FUNCTION_BLOCK CmdSludgeDischargeSLBLogic (* CAT Function Block Type *)
  (* Standard: 61499-2 *)
  (* Version 4.1, 9/30/2026, Claude/Hidryco, Schneider Electric, Rev4.1 - Velocidade reenviada a cada mudanca de comando das bombas e a cada 1 s (SpeedGate aberto); Rev4 - PID pela logica; Rev3.1 - SpeedGate *)
  PACKAGE SE.Nereda;
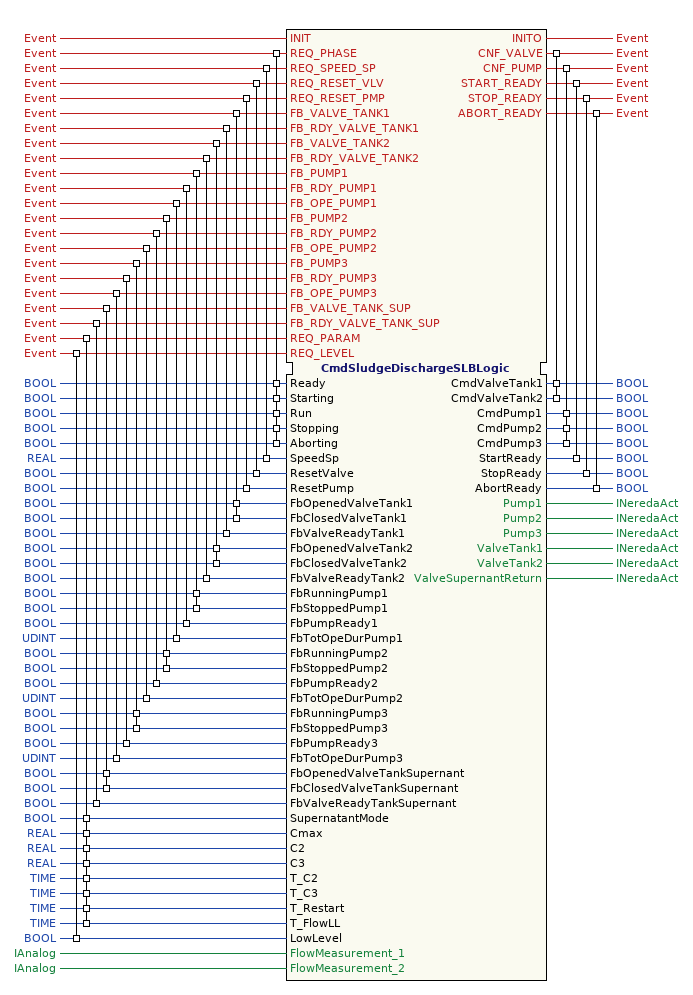
  EVENT_INPUT
    INIT;
    REQ_PHASE WITH Ready, Starting, Run, Stopping, Aborting;
    REQ_SPEED_SP WITH SpeedSp;
    REQ_RESET_VLV WITH ResetValve;
    REQ_RESET_PMP WITH ResetPump;
    FB_VALVE_TANK1 WITH FbOpenedValveTank1, FbClosedValveTank1;
    FB_RDY_VALVE_TANK1 WITH FbValveReadyTank1;
    FB_VALVE_TANK2 WITH FbOpenedValveTank2, FbClosedValveTank2;
    FB_RDY_VALVE_TANK2 WITH FbValveReadyTank2;
    FB_PUMP1 WITH FbRunningPump1, FbStoppedPump1;
    FB_RDY_PUMP1 WITH FbPumpReady1;
    FB_OPE_PUMP1 WITH FbTotOpeDurPump1;
    FB_PUMP2 WITH FbRunningPump2, FbStoppedPump2;
    FB_RDY_PUMP2 WITH FbPumpReady2;
    FB_OPE_PUMP2 WITH FbTotOpeDurPump2;
    FB_PUMP3 WITH FbRunningPump3, FbStoppedPump3;
    FB_RDY_PUMP3 WITH FbPumpReady3;
    FB_OPE_PUMP3 WITH FbTotOpeDurPump3;
    FB_VALVE_TANK_SUP WITH FbOpenedValveTankSupernant, FbClosedValveTankSupernant;
    FB_RDY_VALVE_TANK_SUP WITH FbValveReadyTankSupernant;
    REQ_PARAM WITH SupernatantMode, Cmax, C2, C3, T_C2, T_C3, T_Restart, T_FlowLL; (* Parametros da logica de bombas e da pausa *)
    REQ_LEVEL WITH LowLevel; (* Nivel L do 49LT0001 *)
  END_EVENT
  EVENT_OUTPUT
    INITO;
    CNF_VALVE WITH CmdValveTank1, CmdValveTank2;
    CNF_PUMP WITH CmdPump1, CmdPump2, CmdPump3;
    START_READY WITH StartReady;
    STOP_READY WITH StopReady;
    ABORT_READY WITH AbortReady;
  END_EVENT
  VAR_INPUT
    Ready : BOOL;
    Starting : BOOL;
    Run : BOOL;
    Stopping : BOOL;
    Aborting : BOOL;
    SpeedSp : REAL;
    ResetValve : BOOL;
    ResetPump : BOOL;
    FbOpenedValveTank1 : BOOL;
    FbClosedValveTank1 : BOOL;
    FbValveReadyTank1 : BOOL;
    FbOpenedValveTank2 : BOOL;
    FbClosedValveTank2 : BOOL;
    FbValveReadyTank2 : BOOL;
    FbRunningPump1 : BOOL;
    FbStoppedPump1 : BOOL;
    FbPumpReady1 : BOOL;
    FbTotOpeDurPump1 : UDINT;
    FbRunningPump2 : BOOL;
    FbStoppedPump2 : BOOL;
    FbPumpReady2 : BOOL;
    FbTotOpeDurPump2 : UDINT;
    FbRunningPump3 : BOOL;
    FbStoppedPump3 : BOOL;
    FbPumpReady3 : BOOL;
    FbTotOpeDurPump3 : UDINT;
    FbOpenedValveTankSupernant : BOOL;
    FbClosedValveTankSupernant : BOOL;
    FbValveReadyTankSupernant : BOOL;
    SupernatantMode : BOOL; (* TRUE = sobrenadante (2 servico + 1 reserva); FALSE/desligado = lodo (1 servico + 2 reserva) *)
    Cmax : REAL; (* Vazao maxima de 1 bomba [m3/h] *)
    C2 : REAL; (* Vazao por bomba na entrada da 2a bomba [m3/h] *)
    C3 : REAL; (* Vazao por bomba abaixo da qual sai 1 bomba [m3/h] *)
    T_C2 : TIME; (* Tempo em C2 *)
    T_C3 : TIME; (* Tempo abaixo de C3 *)
    T_Restart : TIME; (* Pausa: tempo para retomar *)
    T_FlowLL : TIME; (* Vazao LL por este tempo com bomba rodando = pausa (0 = desabilitado) *)
    LowLevel : BOOL; (* Nivel L do 49LT0001 (pausa a descarga) *)
  END_VAR
  VAR_OUTPUT
    CmdValveTank1 : BOOL;
    CmdValveTank2 : BOOL;
    CmdPump1 : BOOL;
    CmdPump2 : BOOL;
    CmdPump3 : BOOL;
    StartReady : BOOL;
    StopReady : BOOL;
    AbortReady : BOOL;
  END_VAR
  SOCKETS
    FlowMeasurement_1 : IAnalog;
  END_SOCKETS
  SOCKETS
    FlowMeasurement_2 : IAnalog;
  END_SOCKETS
  PLUGS
    Pump1 : INeredaAct;
    Pump2 : INeredaAct;
    Pump3 : INeredaAct;
    ValveTank1 : INeredaAct;
    ValveTank2 : INeredaAct;
    ValveSupernantReturn : INeredaAct;
  END_PLUGS
  (* 01 - FUNCTIONNAL INPUT INTERFACE *)
  (* 00 - INITIALIZATION *)
  (* 05 - LOGIC *)
  (* 06 - HMI INTERFACE *)
  (* 03 - FIELD INTERFACE *)
  (* 02 - FUNCTIONNAL OUTPUT INTERFACE *)
  (* Command Logic *)
  (* SIGNAL SELECTION *)
  FBS
    CmdLogic : CmdSludgeDischargeSLBLogicBasic;
    ValveCmdSmoothTank1 : boolValueChanged;
    PumpCmdSmooth1 : boolValueChanged;
    FbOpenValveTank1 : DS_SELECTX_2536758B411A6CE51; {SET_ATTRIBUTE(Configuration.GenericFBType.InterfaceParams, Runtime.Standard#CNTX:=2;CNTY:=1;DI${CNTX,_,CNTY$}:BOOL)}
    FbCloseValveTank1 : DS_SELECTX_2536758B411A6CE51; {SET_ATTRIBUTE(Configuration.GenericFBType.InterfaceParams, Runtime.Standard#CNTX:=2;CNTY:=1;DI${CNTX,_,CNTY$}:BOOL)}
    FbRunPump1 : DS_SELECTX_2536758B411A6CE51; {SET_ATTRIBUTE(Configuration.GenericFBType.InterfaceParams, Runtime.Standard#CNTX:=2;CNTY:=1;DI${CNTX,_,CNTY$}:BOOL)}
    FbStopPump1 : DS_SELECTX_2536758B411A6CE51; {SET_ATTRIBUTE(Configuration.GenericFBType.InterfaceParams, Runtime.Standard#CNTX:=2;CNTY:=1;DI${CNTX,_,CNTY$}:BOOL)}
    FbReadyPump1 : DS_SELECTX_2536758B411A6CE51; {SET_ATTRIBUTE(Configuration.GenericFBType.InterfaceParams, Runtime.Standard#CNTX:=2;CNTY:=1;DI${CNTX,_,CNTY$}:BOOL)}
    FbReadyValveTank1 : DS_SELECTX_2536758B411A6CE51; {SET_ATTRIBUTE(Configuration.GenericFBType.InterfaceParams, Runtime.Standard#CNTX:=2;CNTY:=1;DI${CNTX,_,CNTY$}:BOOL)}
    ValveCmdTank1 : BOOL2INT;
    PumpCmd1 : BOOL2INT;
    FbTotOpePump1 : DS_SELECTX_29841900CAFD143A; {SET_ATTRIBUTE(Configuration.GenericFBType.InterfaceParams, Runtime.Standard#CNTX:=2;CNTY:=1;DI${CNTX,_,CNTY$}:UDINT)}
    FbRunPump2 : DS_SELECTX_2536758B411A6CE51; {SET_ATTRIBUTE(Configuration.GenericFBType.InterfaceParams, Runtime.Standard#CNTX:=2;CNTY:=1;DI${CNTX,_,CNTY$}:BOOL)}
    FbStopPump2 : DS_SELECTX_2536758B411A6CE51; {SET_ATTRIBUTE(Configuration.GenericFBType.InterfaceParams, Runtime.Standard#CNTX:=2;CNTY:=1;DI${CNTX,_,CNTY$}:BOOL)}
    FbReadyPump2 : DS_SELECTX_2536758B411A6CE51; {SET_ATTRIBUTE(Configuration.GenericFBType.InterfaceParams, Runtime.Standard#CNTX:=2;CNTY:=1;DI${CNTX,_,CNTY$}:BOOL)}
    FbTotOpePump2 : DS_SELECTX_29841900CAFD143A; {SET_ATTRIBUTE(Configuration.GenericFBType.InterfaceParams, Runtime.Standard#CNTX:=2;CNTY:=1;DI${CNTX,_,CNTY$}:UDINT)}
    FbRunPump3 : DS_SELECTX_2536758B411A6CE51; {SET_ATTRIBUTE(Configuration.GenericFBType.InterfaceParams, Runtime.Standard#CNTX:=2;CNTY:=1;DI${CNTX,_,CNTY$}:BOOL)}
    FbStopPump3 : DS_SELECTX_2536758B411A6CE51; {SET_ATTRIBUTE(Configuration.GenericFBType.InterfaceParams, Runtime.Standard#CNTX:=2;CNTY:=1;DI${CNTX,_,CNTY$}:BOOL)}
    FbReadyPump3 : DS_SELECTX_2536758B411A6CE51; {SET_ATTRIBUTE(Configuration.GenericFBType.InterfaceParams, Runtime.Standard#CNTX:=2;CNTY:=1;DI${CNTX,_,CNTY$}:BOOL)}
    FbTotOpePump3 : DS_SELECTX_29841900CAFD143A; {SET_ATTRIBUTE(Configuration.GenericFBType.InterfaceParams, Runtime.Standard#CNTX:=2;CNTY:=1;DI${CNTX,_,CNTY$}:UDINT)}
    FbOpenValveTank2 : DS_SELECTX_2536758B411A6CE51; {SET_ATTRIBUTE(Configuration.GenericFBType.InterfaceParams, Runtime.Standard#CNTX:=2;CNTY:=1;DI${CNTX,_,CNTY$}:BOOL)}
    FbCloseValveTank2 : DS_SELECTX_2536758B411A6CE51; {SET_ATTRIBUTE(Configuration.GenericFBType.InterfaceParams, Runtime.Standard#CNTX:=2;CNTY:=1;DI${CNTX,_,CNTY$}:BOOL)}
    FbReadyValveTank2 : DS_SELECTX_2536758B411A6CE51; {SET_ATTRIBUTE(Configuration.GenericFBType.InterfaceParams, Runtime.Standard#CNTX:=2;CNTY:=1;DI${CNTX,_,CNTY$}:BOOL)}
    ValveCmdSmoothTank2 : boolValueChanged;
    ValveCmdTank2 : BOOL2INT;
    PumpCmdSmooth2 : boolValueChanged;
    PumpCmd2 : BOOL2INT;
    PumpCmdSmooth3 : boolValueChanged;
    PumpCmd3 : BOOL2INT;
    MergeValveCmd : E_MERGE;
    MergePumpCmd : E_MERGE;
    IThis : CmdSludgeDischargeSLBLogic_HMI(QI := TRUE);
    PID : PID; {SET_ATTRIBUTE(Configuration.Component.HideUnusedPorts, )}
    PIDISc : PID_Manager;
    SpeedSp1 : SpeedSpFlowSensorFail;
    Flow_Status : decodeStatus; {SET_ATTRIBUTE(Configuration.Component.HideUnusedPorts, )}
    OR1 : OR_550FE6D62F509EB3; {SET_ATTRIBUTE(Configuration.GenericFBType.InterfaceParams, Runtime.Standard#CNT:=3;OUT:BOOL)}
    PumpCmdSmooth4 : boolValueChanged;
    PumpCmd4 : BOOL2INT;
    FbOpenValveTankSupernant : DS_SELECTX_2536758B411A6CE51; {SET_ATTRIBUTE(Configuration.GenericFBType.InterfaceParams, Runtime.Standard#CNTX:=2;CNTY:=1;DI${CNTX,_,CNTY$}:BOOL)}
    FbCloseValveTankSupernant : DS_SELECTX_2536758B411A6CE51; {SET_ATTRIBUTE(Configuration.GenericFBType.InterfaceParams, Runtime.Standard#CNTX:=2;CNTY:=1;DI${CNTX,_,CNTY$}:BOOL)}
    FbReadyValveTankSupernant : DS_SELECTX_2536758B411A6CE51; {SET_ATTRIBUTE(Configuration.GenericFBType.InterfaceParams, Runtime.Standard#CNTX:=2;CNTY:=1;DI${CNTX,_,CNTY$}:BOOL)}
    TickCycle : E_CYCLE(DT := T#1s);
    SpeedGate : E_PERMIT;
  END_FBS
  EVENT_CONNECTIONS
    FbOpenValveTank1.CNF1 TO FbCloseValveTank1.REQ1;
    FbOpenValveTank1.CNF2 TO FbCloseValveTank1.REQ2;
    FbRunPump1.CNF1 TO FbStopPump1.REQ1;
    FbRunPump1.CNF2 TO FbStopPump1.REQ2;
    ValveCmdSmoothTank1.CHD TO ValveCmdTank1.DD5870AA881150BB;
    PumpCmdSmooth1.CHD TO PumpCmd1.DD5870AA881150BB;
    FB_VALVE_TANK1 TO FbOpenValveTank1.REQ2;
    FB_PUMP1 TO FbRunPump1.REQ2;
    FB_RDY_VALVE_TANK1 TO FbReadyValveTank1.REQ2;
    FB_RDY_PUMP1 TO FbReadyPump1.REQ2;
    REQ_PHASE TO CmdLogic.READY;
    REQ_PHASE TO CmdLogic.STARTING;
    REQ_PHASE TO CmdLogic.RUN;
    REQ_PHASE TO CmdLogic.STOPPING;
    REQ_PHASE TO CmdLogic.ABORTING;
    FbCloseValveTank1.IND TO CmdLogic.VALVE_FB_OPEN;
    FbStopPump1.IND TO CmdLogic.PUMP_FB_RUN;
    FbReadyValveTank1.IND TO CmdLogic.VALVE_AVAILABLE;
    FbReadyPump1.IND TO CmdLogic.PUMP_NO_AVAILABLE;
    CmdLogic.VALVE_CNF TO ValveCmdSmoothTank1.REQ;
    CmdLogic.PUMP_CNF TO PumpCmdSmooth1.REQ;
    CmdLogic.START_READY TO START_READY;
    CmdLogic.STOP_READY TO STOP_READY;
    CmdLogic.ABORTED_READY TO ABORT_READY;
    FbRunPump2.CNF1 TO FbStopPump2.REQ1;
    FbRunPump2.CNF2 TO FbStopPump2.REQ2;
    FbRunPump3.CNF1 TO FbStopPump3.REQ1;
    FbRunPump3.CNF2 TO FbStopPump3.REQ2;
    FbOpenValveTank2.CNF1 TO FbCloseValveTank2.REQ1;
    FbOpenValveTank2.CNF2 TO FbCloseValveTank2.REQ2;
    ValveCmdSmoothTank2.CHD TO ValveCmdTank2.DD5870AA881150BB;
    PumpCmdSmooth2.CHD TO PumpCmd2.DD5870AA881150BB;
    PumpCmdSmooth3.CHD TO PumpCmd3.DD5870AA881150BB;
    FbReadyValveTank2.IND TO CmdLogic.VALVE_AVAILABLE;
    FbCloseValveTank2.IND TO CmdLogic.VALVE_FB_OPEN;
    FbTotOpePump1.IND TO CmdLogic.51724FB542235B99;
    FbTotOpePump3.IND TO CmdLogic.51724FB542235B99;
    FbTotOpePump2.IND TO CmdLogic.51724FB542235B99;
    FbStopPump3.IND TO CmdLogic.PUMP_FB_RUN;
    FbStopPump2.IND TO CmdLogic.PUMP_FB_RUN;
    FbReadyPump2.IND TO CmdLogic.PUMP_NO_AVAILABLE;
    FbReadyPump3.IND TO CmdLogic.PUMP_NO_AVAILABLE;
    FB_RDY_VALVE_TANK2 TO FbReadyValveTank2.REQ2;
    FB_VALVE_TANK2 TO FbOpenValveTank2.REQ2;
    FB_RDY_PUMP3 TO FbReadyPump3.REQ2;
    FB_OPE_PUMP3 TO FbTotOpePump3.REQ2;
    FB_PUMP3 TO FbRunPump3.REQ2;
    FB_RDY_PUMP2 TO FbReadyPump2.REQ2;
    FB_OPE_PUMP2 TO FbTotOpePump2.REQ2;
    FB_PUMP2 TO FbRunPump2.REQ2;
    ValveTank1.CC753684FA882790 TO FbReadyValveTank1.REQ1;
    ValveTank1.9CD053F8408797ED TO FbOpenValveTank1.REQ1;
    ValveTank2.9CD053F8408797ED TO FbOpenValveTank2.REQ1;
    ValveTank2.CC753684FA882790 TO FbReadyValveTank2.REQ1;
    Pump1.2DA8AEC15204E92D TO FbTotOpePump1.REQ1;
    Pump1.CC753684FA882790 TO FbReadyPump1.REQ1;
    Pump1.9CD053F8408797ED TO FbRunPump1.REQ1;
    FB_OPE_PUMP1 TO FbTotOpePump1.REQ2;
    Pump2.9CD053F8408797ED TO FbRunPump2.REQ1;
    Pump2.CC753684FA882790 TO FbReadyPump2.REQ1;
    Pump2.2DA8AEC15204E92D TO FbTotOpePump2.REQ1;
    Pump3.9CD053F8408797ED TO FbRunPump3.REQ1;
    Pump3.CC753684FA882790 TO FbReadyPump3.REQ1;
    Pump3.2DA8AEC15204E92D TO FbTotOpePump3.REQ1;
    ValveCmdTank1.6FC99A5BD1C38561 TO ValveTank1.0F1CDF9A9B4A227A;
    ValveCmdTank2.6FC99A5BD1C38561 TO ValveTank2.0F1CDF9A9B4A227A;
    PumpCmd1.6FC99A5BD1C38561 TO Pump1.0F1CDF9A9B4A227A;
    PumpCmd2.6FC99A5BD1C38561 TO Pump2.0F1CDF9A9B4A227A;
    PumpCmd3.6FC99A5BD1C38561 TO Pump3.0F1CDF9A9B4A227A;
    CmdLogic.PUMP_CNF TO PumpCmdSmooth3.REQ;
    CmdLogic.PUMP_CNF TO PumpCmdSmooth2.REQ;
    CmdLogic.VALVE_CNF TO ValveCmdSmoothTank2.REQ;
    REQ_RESET_VLV TO Pump3.37BBC1F841739733;
    REQ_RESET_VLV TO Pump1.37BBC1F841739733;
    REQ_RESET_VLV TO Pump2.37BBC1F841739733;
    ValveCmdSmoothTank1.CHD TO MergeValveCmd.EI1;
    ValveCmdSmoothTank2.CHD TO MergeValveCmd.EI2;
    MergeValveCmd.EO TO CNF_VALVE;
    PumpCmdSmooth1.CHD TO MergePumpCmd.EI1;
    PumpCmdSmooth2.CHD TO MergePumpCmd.EI2;
    PumpCmdSmooth3.CHD TO MergePumpCmd.EI2;
    MergePumpCmd.EO TO CNF_PUMP;
    PIDISc.CE80458C9D5EF15A TO INITO;
    FlowMeasurement_1.REQ TO Flow_Status.REQ;
    PumpCmdSmooth3.CHD TO OR1.REQ;
    PumpCmdSmooth2.CHD TO OR1.REQ;
    PumpCmdSmooth1.CHD TO OR1.REQ;
    OR1.CNF TO PIDISc.REQ;
    FlowMeasurement_1.REQ TO SpeedSp1.B5D6B08FA2666F02;
    INIT TO IThis.2F65FBA3287455C1;
    CmdLogic.001688431DB935DE TO IThis.2568B13DF8BCDE7D;
    IThis.FFFD39D6E5C086B9 TO PIDISc.INIT;
    Flow_Status.CNF TO SpeedSp1.B5D6B08FA2666F02;
    PumpCmdSmooth4.CHD TO PumpCmd4.DD5870AA881150BB;
    PumpCmd4.6FC99A5BD1C38561 TO ValveSupernantReturn.0F1CDF9A9B4A227A;
    CmdLogic.VALVE_CNF TO PumpCmdSmooth4.REQ;
    FbOpenValveTankSupernant.CNF1 TO FbCloseValveTankSupernant.REQ1;
    FbOpenValveTankSupernant.CNF2 TO FbCloseValveTankSupernant.REQ2;
    ValveSupernantReturn.CC753684FA882790 TO FbReadyValveTankSupernant.REQ2;
    ValveSupernantReturn.9CD053F8408797ED TO FbOpenValveTankSupernant.REQ2;
    FB_VALVE_TANK_SUP TO FbOpenValveTankSupernant.REQ1;
    FB_RDY_VALVE_TANK_SUP TO FbReadyValveTankSupernant.REQ1;
    FbReadyValveTankSupernant.IND TO CmdLogic.VALVE_AVAILABLE;
    FbCloseValveTankSupernant.IND TO CmdLogic.VALVE_FB_OPEN;
    REQ_RESET_PMP TO ValveSupernantReturn.37BBC1F841739733;
    IThis.FFFD39D6E5C086B9 TO TickCycle.START;
    TickCycle.EO TO CmdLogic.2AFCCC4D006C5A58;
    REQ_SPEED_SP TO CmdLogic.888C7FFA93152C07;
    REQ_PARAM TO CmdLogic.888C7FFA93152C07;
    CmdLogic.948C0A3C8D4A59E4 TO PIDISc.REQ;
    CmdLogic.948C0A3C8D4A59E4 TO SpeedSp1.B5D6B08FA2666F02;
    REQ_LEVEL TO CmdLogic.19EED5631A4ADE11;
    FlowMeasurement_1.REQ_STATUS TO Flow_Status.REQ;
    Flow_Status.CNF TO CmdLogic.E12F00872D66F11F;
    SpeedSp1.1FEAADE7145F64BE TO SpeedGate.EI;
    SpeedGate.EO TO Pump1.1E00729184986247;
    SpeedGate.EO TO Pump2.1E00729184986247;
    SpeedGate.EO TO Pump3.1E00729184986247;
    SpeedGate.EO TO ValveSupernantReturn.1E00729184986247;
    PID.CNF TO CmdLogic.D9E0400EF0DD670E;
    CmdLogic.6F9F08BA58B8009D TO SpeedSp1.B5D6B08FA2666F02;
    OR1.CNF TO SpeedSp1.B5D6B08FA2666F02;
    TickCycle.EO TO SpeedSp1.B5D6B08FA2666F02;
  END_CONNECTIONS
  DATA_CONNECTIONS
    ValveCmdSmoothTank1.Output TO ValveCmdTank1.4573FC8F228EB71D;
    PumpCmdSmooth1.Output TO PumpCmd1.4573FC8F228EB71D;
    ValveCmdSmoothTank1.Output TO CmdValveTank1;
    PumpCmdSmooth1.Output TO CmdPump1;
    FbOpenedValveTank1 TO FbOpenValveTank1.DI2_1;
    FbClosedValveTank1 TO FbCloseValveTank1.DI2_1;
    FbRunningPump1 TO FbRunPump1.DI2_1;
    FbStoppedPump1 TO FbStopPump1.DI2_1;
    FbValveReadyTank1 TO FbReadyValveTank1.DI2_1;
    FbPumpReady1 TO FbReadyPump1.DI2_1;
    Ready TO CmdLogic.Ready;
    Starting TO CmdLogic.Starting;
    Run TO CmdLogic.RunningState;
    Stopping TO CmdLogic.Stopping;
    Aborting TO CmdLogic.Aborting;
    CmdLogic.StartReady TO StartReady;
    CmdLogic.StopReady TO StopReady;
    CmdLogic.AbortedReady TO AbortReady;
    ValveCmdSmoothTank2.Output TO ValveCmdTank2.4573FC8F228EB71D;
    PumpCmdSmooth2.Output TO PumpCmd2.4573FC8F228EB71D;
    PumpCmdSmooth3.Output TO PumpCmd3.4573FC8F228EB71D;
    FbOpenValveTank1.OUT1 TO CmdLogic.EE3E325E38DB6D95;
    FbCloseValveTank1.OUT1 TO CmdLogic.4E0EDF1D6602AD7F;
    FbReadyValveTank1.OUT1 TO CmdLogic.78D1EE87F8AE3968;
    FbOpenValveTank2.OUT1 TO CmdLogic.38A9A390455B9A4F;
    FbCloseValveTank2.OUT1 TO CmdLogic.9C68F1DF546D3052;
    FbReadyValveTank2.OUT1 TO CmdLogic.71509D151A182356;
    FbRunPump1.OUT1 TO CmdLogic.41857D3371CE356D;
    FbStopPump1.OUT1 TO CmdLogic.8966D3D93AE9B840;
    FbReadyPump1.OUT1 TO CmdLogic.92B7B9D369930721;
    FbTotOpePump1.OUT1 TO CmdLogic.0D663C311D386D2A;
    FbRunPump2.OUT1 TO CmdLogic.450E1E0E9DC1B17B;
    FbRunPump3.OUT1 TO CmdLogic.C4E5F519898D3848;
    FbStopPump2.OUT1 TO CmdLogic.EE227D743F972C8D;
    FbStopPump3.OUT1 TO CmdLogic.956E0A0A54836360;
    FbReadyPump2.OUT1 TO CmdLogic.8294BD3E31844391;
    FbReadyPump3.OUT1 TO CmdLogic.0EC6936CA60DF719;
    FbTotOpePump2.OUT1 TO CmdLogic.57AA0C889DBD9CF5;
    FbTotOpePump3.OUT1 TO CmdLogic.5E64FC3A91DBC3F6;
    FbClosedValveTank2 TO FbCloseValveTank2.DI2_1;
    FbOpenedValveTank2 TO FbOpenValveTank2.DI2_1;
    FbValveReadyTank2 TO FbReadyValveTank2.DI2_1;
    FbPumpReady3 TO FbReadyPump3.DI2_1;
    FbTotOpeDurPump3 TO FbTotOpePump3.DI2_1;
    FbStoppedPump3 TO FbStopPump3.DI2_1;
    FbRunningPump3 TO FbRunPump3.DI2_1;
    FbTotOpeDurPump2 TO FbTotOpePump2.DI2_1;
    FbPumpReady2 TO FbReadyPump2.DI2_1;
    FbRunningPump2 TO FbRunPump2.DI2_1;
    FbStoppedPump2 TO FbStopPump2.DI2_1;
    ValveTank1.7F6CC7FEB9223DF3 TO FbOpenValveTank1.DI1_1;
    ValveTank1.A8D6C4A1FDCCA991 TO FbCloseValveTank1.DI1_1;
    ValveTank1.8A8A07EFCDA1443C TO FbReadyValveTank1.DI1_1;
    ValveTank2.8A8A07EFCDA1443C TO FbReadyValveTank2.DI1_1;
    ValveTank2.A8D6C4A1FDCCA991 TO FbCloseValveTank2.DI1_1;
    ValveTank2.7F6CC7FEB9223DF3 TO FbOpenValveTank2.DI1_1;
    Pump1.B762734C094A7162 TO FbRunPump1.DI1_1;
    Pump1.D83B5BDEFA4D797C TO FbStopPump1.DI1_1;
    Pump1.8A8A07EFCDA1443C TO FbReadyPump1.DI1_1;
    Pump1.C7F638DBF6B860D2 TO FbTotOpePump1.DI1_1;
    FbTotOpeDurPump1 TO FbTotOpePump1.DI2_1;
    Pump2.B762734C094A7162 TO FbRunPump2.DI1_1;
    Pump2.D83B5BDEFA4D797C TO FbStopPump2.DI1_1;
    Pump2.8A8A07EFCDA1443C TO FbReadyPump2.DI1_1;
    Pump2.C7F638DBF6B860D2 TO FbTotOpePump2.DI1_1;
    Pump3.C7F638DBF6B860D2 TO FbTotOpePump3.DI1_1;
    Pump3.D83B5BDEFA4D797C TO FbStopPump3.DI1_1;
    Pump3.B762734C094A7162 TO FbRunPump3.DI1_1;
    Pump3.8A8A07EFCDA1443C TO FbReadyPump3.DI1_1;
    ValveCmdTank1.A6DEF5F9C27C1848 TO ValveTank1.710D7FC54EE3F35A;
    ValveCmdTank2.A6DEF5F9C27C1848 TO ValveTank2.710D7FC54EE3F35A;
    PumpCmd1.A6DEF5F9C27C1848 TO Pump1.710D7FC54EE3F35A;
    PumpCmd2.A6DEF5F9C27C1848 TO Pump2.710D7FC54EE3F35A;
    PumpCmd3.A6DEF5F9C27C1848 TO Pump3.710D7FC54EE3F35A;
    CmdLogic.AB3759E05952DF13 TO ValveCmdSmoothTank1.Input;
    CmdLogic.1F14A2AEE3E323F8 TO ValveCmdSmoothTank2.Input;
    CmdLogic.945BF4FE52310595 TO PumpCmdSmooth1.Input;
    CmdLogic.750D687533E86DDC TO PumpCmdSmooth2.Input;
    CmdLogic.A7428AB4F66CF0EA TO PumpCmdSmooth3.Input;
    ResetValve TO Pump2.EA28053F07575F36;
    ResetValve TO Pump3.EA28053F07575F36;
    ResetValve TO Pump1.EA28053F07575F36;
    ValveCmdSmoothTank2.Output TO CmdValveTank2;
    PumpCmdSmooth2.Output TO CmdPump2;
    PumpCmdSmooth3.Output TO CmdPump3;
    FlowMeasurement_1.Status TO Flow_Status.Status;
    Flow_Status.FailAlarm TO SpeedSp1.1C28FEF37A13F67F;
    FlowMeasurement_1.ValueMin TO SpeedSp1.B08827D02DBBFA97;
    FlowMeasurement_1.ValueMax TO SpeedSp1.75C86D8B7647050C;
    PumpCmdSmooth1.Output TO OR1.IN1;
    PumpCmdSmooth2.Output TO OR1.IN2;
    PumpCmdSmooth3.Output TO OR1.IN3;
    OR1.OUT TO PIDISc.RunPID;
    CmdLogic.DB4AE032AE08C110 TO IThis.930FFC0215E780EF;
    SpeedSp1.87931CA83794BFFD TO Pump3.1BC103921BBFDA0B;
    SpeedSp1.87931CA83794BFFD TO Pump2.1BC103921BBFDA0B;
    SpeedSp1.87931CA83794BFFD TO Pump1.1BC103921BBFDA0B;
    PumpCmdSmooth4.Output TO PumpCmd4.4573FC8F228EB71D;
    PumpCmd4.A6DEF5F9C27C1848 TO ValveSupernantReturn.710D7FC54EE3F35A;
    CmdLogic.56F564B55D225FAF TO PumpCmdSmooth4.Input;
    SpeedSp1.87931CA83794BFFD TO ValveSupernantReturn.1BC103921BBFDA0B;
    ValveSupernantReturn.8A8A07EFCDA1443C TO FbReadyValveTankSupernant.DI2_1;
    ValveSupernantReturn.7F6CC7FEB9223DF3 TO FbOpenValveTankSupernant.DI2_1;
    ValveSupernantReturn.A8D6C4A1FDCCA991 TO FbCloseValveTankSupernant.DI2_1;
    FbOpenedValveTankSupernant TO FbOpenValveTankSupernant.DI1_1;
    FbClosedValveTankSupernant TO FbCloseValveTankSupernant.DI1_1;
    FbValveReadyTankSupernant TO FbReadyValveTankSupernant.DI1_1;
    FbOpenValveTankSupernant.OUT1 TO CmdLogic.8A3A0D8C0A296294;
    FbCloseValveTankSupernant.OUT1 TO CmdLogic.5AB763DA99D1722E;
    FbReadyValveTankSupernant.OUT1 TO CmdLogic.C2A6AEC1BFED4499;
    ResetPump TO ValveSupernantReturn.EA28053F07575F36;
    SpeedSp TO CmdLogic.38A57B28987BAE06;
    SupernatantMode TO CmdLogic.B8EE5B594802026A;
    Cmax TO CmdLogic.0A323B5BB10D6790;
    C2 TO CmdLogic.7B6FA0EADBC872E0;
    C3 TO CmdLogic.FBBD66E4176C0F4A;
    T_C2 TO CmdLogic.2EE8E2AD063EE95E;
    T_C3 TO CmdLogic.097CEF7D3109D4BE;
    T_Restart TO CmdLogic.37F2A16CD48B9A9D;
    T_FlowLL TO CmdLogic.E9499B195D781C20;
    CmdLogic.CFFB125A7B539DE2 TO PIDISc.Setpoint;
    CmdLogic.CFFB125A7B539DE2 TO SpeedSp1.3BE251DFC2E7905D;
    LowLevel TO CmdLogic.E364687AE6285E4B;
    Flow_Status.LoLoAlarm TO CmdLogic.CF4621EC925C43E9;
    Flow_Status.FailAlarm TO CmdLogic.F66FAF9E12E91CF7;
    OR1.OUT TO SpeedGate.PERMIT;
    PID.Out TO CmdLogic.A7D276693781888D;
    CmdLogic.1E314D8B4487BA0C TO SpeedSp1.4727B0C2E5DD09FB;
  END_CONNECTIONS
  ADAPTER_CONNECTIONS
    PIDISc.FACD1DD4E791A86A TO PID.ISc;
    FlowMeasurement_2 TO PID.IPv;
  END_CONNECTIONS
END_FUNCTION_BLOCK
